TYPE
    ST_MediatorInterface : STRUCT
        Request    : BOOL;
        Permission : BOOL;
    END_STRUCT
END_TYPE

(* stored: Version 1.1.0.1
   DUT ST_MediatorInterface: Id {02ccfe20-b771-4dd1-9dbf-a71b06eda2a1} *)
